{attribute 'GeneratedUsingTerminal: EL6720-0000-0016'}
{attribute addProperty BoxType "EL6720-0000-0016"}
{attribute addProperty Id "InfoDataAT %I*InfoData_41C547A32"}
{attribute addProperty CRC "3204926373"}
{attribute addProperty Size "2"}
TYPE EL6720_BF074BA5 EXTENDS EtcSlaveTerminalBase_947E5A46 :
STRUCT
	{attribute addProperty Name "InfoData"}
	InfoData : InfoData_41C547A3;
END_STRUCT
END_TYPE

(* stored: Version 1.2.0.0, ProductVersion 3.1.4024.9
   DUT EL6720_BF074BA5: Id {8f2d4cea-ef23-4b35-a933-2691a02d7b81} *)
